FUNCTION_BLOCK F_SHL (* shift left *)
  PACKAGE iec61131::arithmetic;
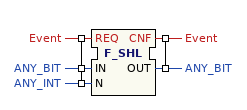
  EVENT_INPUT
    REQ WITH IN, N; (* Service Request *)
  END_EVENT
  EVENT_OUTPUT
    CNF WITH OUT; (* Confirmation of Requested Service *)
  END_EVENT
  VAR_INPUT
    IN : ANY_BIT; (* left-shifted *)
    N : ANY_INT; (* left-shifted by N bits *)
  END_VAR
  VAR_OUTPUT
    OUT : ANY_BIT; (* left-shifted by N zero-filled on right *)
  END_VAR
END_FUNCTION_BLOCK
